FUNCTION_BLOCK FB_RollingAverage
VAR
    samples : ARRAY[0..15] OF INT;
    sampleCount : INT := 8;
    nextIndex : INT;
END_VAR

METHOD Step : INT
VAR_INPUT
    sample : INT;
END_VAR
VAR
    sum : DINT;
    i : INT;
END_VAR
samples[nextIndex] := sample;
nextIndex := (nextIndex + 1) MOD sampleCount;
sum := 0;
FOR i := 1 TO sampleCount DO
    sum := sum + samples[i];
END_FOR
Step := DINT_TO_INT(sum / sampleCount);
END_METHOD

END_FUNCTION_BLOCK

(* stored: Version 1.1.0.1
   POU FB_RollingAverage: Id {41e4f492-3ae5-498c-b8ff-a39c88c63647}, SpecialFunc None
   Method Step: Id {c174831a-9762-45b7-8b37-6479933673af} *)
